// TIA Portal V20 export
// export: Created 2025-12-01T14:57:12.2354919Z, ExportSetting None, DisplayName Totally Integrated Automation Portal, DisplayVersion V20 Update 3, DisplayName TIA Portal Openness, DisplayVersion V20 Update 3, DisplayName TIA Portal Version Control Interface, DisplayVersion V20 Update 3, DisplayName STEP 7 Professional, DisplayVersion V20 Update 3, DisplayName STEP 7 Safety, DisplayVersion V20 Update 2, DisplayName WinCC Basic/Comfort/Advanced, DisplayVersion V20 Update 3, DisplayName WinCC Professional, DisplayVersion V20 Update 3, DisplayName WinCC Unified, DisplayVersion V20 Update 3
FUNCTION "FC993_CTRL_VAR_Lenze_i550_ASi" : Void   // FC993, LAD
{ S7_Optimized_Access := 'TRUE' }
// M.Familiar: Adaptado al nuevo base 14_02_2023.
// stored: AutoNumber false, SetENOAutomatically false
   VAR_INPUT
      DIR_INI_NODO : Int;   // Direccion inicial Gateway
      Num_Motor : Int;   // Numero de motor
      Avance : Bool;
      Retroceso : Bool;
      Rearme : Bool;   // Rearme variador
      Conexion_Estrella : Bool;
      Motor_2 : Bool;
      Sentido_Giro : Bool;   // Sentido giro
      "Activar Salida Digital DO1" : Bool;   // Activar Salida DO1
      Consigna_FR : Word;   // Consigna
   END_VAR
   VAR_TEMP
      ByteOffset : Int;
      Codigo_Area_Lectura : Byte;
      Codigo_Area_Escritura : Byte;
      Byte1_Status_Variador : Byte;
      Byte2_Status_Variador : Byte;
      Byte1PalabraControl : Byte;
      Byte2PalabraControl : Byte;
      Num_SETUP : Int;   // 1-triangulo Motor1/ 2-triangulo Motor 2 / 3-Estrella Motor1/4-Estrella Motor 2
   END_VAR
   VAR CONSTANT
      Area_SCR_DB : Byte := 16#84;
   END_VAR
BEGIN

REGION Network 1 (SCL): Simulador on?
   IF "Activar_Simulador" THEN
       #Codigo_Area_Lectura := 16#81;     // Area entradas %I
       #Codigo_Area_Escritura := 16#82;  // Area salidas %Q
   ELSE
       #Codigo_Area_Lectura := 16#1;     // Area entradas periferia 
       #Codigo_Area_Escritura := 16#2;  // Area salidas periferia 
   END_IF;
END_REGION

REGION Network 2 (SCL): Calcular Direccion inicial del nodo
   // M.FAMILIAR : Cambio calculo inicial de Byteoffset en base a direccion inicial de GATEWAY por directamnete direccion inicial del nodo del motor.
   REGION  //Definicion de direcciones a tratar//
       #ByteOffset := #DIR_INI_NODO;   

   END_REGION
END_REGION

REGION Network 3 (SCL): Lectura variador >>PLC
   REGION // lectura Status Variador    

       #Byte2_Status_Variador := PEEK_BYTE(area := #Codigo_Area_Lectura, dbNumber := 0, byteOffset := #ByteOffset);  //Leemos segundo Byte del status variador.
       POKE(area := #Area_SCR_DB,                                //Definimos tipo de area de memoria de escritura, en este caso un DB.
            dbNumber := 941,                                    //Ponemos 0 si es area de E/S si no ponemos numero de DB.
            byteOffset := (#Num_Motor * 18 - 17),                  // Definimos offset de Byte donde queremos escribir.
            value := #Byte2_Status_Variador,                 // valor que queremos escribir en destino.
            ENO => ENO);                                       // Consulta de ejecucion.
       #Byte1_Status_Variador := PEEK_BYTE(area := #Codigo_Area_Lectura, dbNumber := 0, byteOffset := #ByteOffset+1);  //Leemos primer Byte del status variador.
       POKE(area := #Area_SCR_DB,                                //Definimos tipo de area de memoria de escritura, en este caso un DB.
            dbNumber := 941,                                    //Ponemos 0 si es area de E/S si no ponemos numero de DB.
            byteOffset := (#Num_Motor* 18 - 18),                  // Definimos offset de Byte donde queremos escribir.
            value := #Byte1_Status_Variador,                 // valor que queremos escribir en destino.
            ENO => ENO);





    //lectura Words de codigo de error y corriente actual motor

       "DB941_Datos_VAR_Lenze_i550_ASi".Lenze_i550[#Num_Motor]."Código de error (Inputs)" := PEEK_WORD (area := #Codigo_Area_Lectura, dbNumber := 0, byteOffset := #ByteOffset + 2);
       "DB941_Datos_VAR_Lenze_i550_ASi".Lenze_i550[#Num_Motor]."Corriente actual (Inputs)" := PEEK_WORD (area := #Codigo_Area_Lectura, dbNumber := 0, byteOffset := #ByteOffset + 4);

    END_REGION
END_REGION

REGION Network 4 (SCL): Seleccion de SetUp Motor
   REGION Selección de juego de parámetros


       // SETUP 1__MOTOR 1 EN "TRIANGULO"
       IF (NOT #Conexion_Estrella AND NOT #Motor_2)
       THEN
           #Num_SETUP := 1;
       END_IF;


       // SETUP 2__MOTOR 2 EN "TRIANGULO"
       IF (NOT #Conexion_Estrella AND #Motor_2)
       THEN
           #Num_SETUP := 2;
       END_IF;


       // SETUP 3__MOTOR 1 EN "ESTRELLA"
       IF (#Conexion_Estrella AND NOT #Motor_2)
       THEN
           #Num_SETUP := 3;
       END_IF;


       // SETUP 4__MOTOR 2 EN "ESTRELLA"
       IF (#Conexion_Estrella AND #Motor_2)
       THEN
           #Num_SETUP := 4;
       END_IF;


   END_REGION




   REGION Ejecución de juego de parámetros

      CASE #Num_SETUP OF
           1:  // SETUP 1  triangulo motor 1 SETUP1
               "DB941_Datos_VAR_Lenze_i550_ASi".Lenze_i550[#Num_Motor]."Palabra de control (Outputs)"."Sel. paramset b0" := FALSE;
               "DB941_Datos_VAR_Lenze_i550_ASi".Lenze_i550[#Num_Motor]."Palabra de control (Outputs)"."Sel. paramset b1" := FALSE;
               ;
           2:  // SETUP 2  triangulo motor 2 SETUP2
               "DB941_Datos_VAR_Lenze_i550_ASi".Lenze_i550[#Num_Motor]."Palabra de control (Outputs)"."Sel. paramset b0" := TRUE;
               "DB941_Datos_VAR_Lenze_i550_ASi".Lenze_i550[#Num_Motor]."Palabra de control (Outputs)"."Sel. paramset b1" := FALSE;
               ;
           3:   // SETUP 3  estrella motor 1 SETUP3
               "DB941_Datos_VAR_Lenze_i550_ASi".Lenze_i550[#Num_Motor]."Palabra de control (Outputs)"."Sel. paramset b0" := FALSE;
               "DB941_Datos_VAR_Lenze_i550_ASi".Lenze_i550[#Num_Motor]."Palabra de control (Outputs)"."Sel. paramset b1" := TRUE;
               ;
          4:   // SETUP 4  estrella motor 2 SETUP4
               "DB941_Datos_VAR_Lenze_i550_ASi".Lenze_i550[#Num_Motor]."Palabra de control (Outputs)"."Sel. paramset b0" := TRUE;
               "DB941_Datos_VAR_Lenze_i550_ASi".Lenze_i550[#Num_Motor]."Palabra de control (Outputs)"."Sel. paramset b1" := TRUE;
               ;
          ELSE  // Si se mete un valor diferente se usa SETUP1
               "DB941_Datos_VAR_Lenze_i550_ASi".Lenze_i550[#Num_Motor]."Palabra de control (Outputs)"."Sel. paramset b0" := FALSE;
               "DB941_Datos_VAR_Lenze_i550_ASi".Lenze_i550[#Num_Motor]."Palabra de control (Outputs)"."Sel. paramset b1" := FALSE;
               ;
       END_CASE;
   END_REGION
END_REGION

REGION Network 5 (SCL): Ejecución de la función

   REGION //Region Control marcha/paro/direccion//
       //Region Control marcha/paro/direccion//

       IF ("DB941_Datos_VAR_Lenze_i550_ASi".Lenze_i550[#Num_Motor]."Estatus variador (Inputs)"."Ready for operation" AND  //Si ready for operation//
           "DB941_Datos_VAR_Lenze_i550_ASi".Lenze_i550[#Num_Motor]."Estatus variador (Inputs)"."Auto setp active" AND      //Si auto setpoint active//     
           NOT "DB941_Datos_VAR_Lenze_i550_ASi".Lenze_i550[#Num_Motor]."Estatus variador (Inputs)"."Fault active") THEN    // si no hay error activo//

           "DB941_Datos_VAR_Lenze_i550_ASi".Lenze_i550[#Num_Motor]."Error activo" := true;                // Activamos Condiciones OK//


           IF (#Avance AND NOT #Retroceso AND NOT #Sentido_Giro)OR ( #Sentido_Giro AND #Retroceso AND NOT #Avance) THEN
               "DB941_Datos_VAR_Lenze_i550_ASi".Lenze_i550[#Num_Motor]."Consigna de frecuencia (Outputs)" := #Consigna_FR;
               "DB941_Datos_VAR_Lenze_i550_ASi".Lenze_i550[#Num_Motor]."Palabra de control (Outputs)"."Run forward" := true;


           ELSE
               IF (NOT #Avance AND #Retroceso AND NOT #Sentido_Giro) OR (#Sentido_Giro AND NOT #Retroceso AND #Avance) THEN
                   "DB941_Datos_VAR_Lenze_i550_ASi".Lenze_i550[#Num_Motor]."Consigna de frecuencia (Outputs)" := #Consigna_FR;
                   "DB941_Datos_VAR_Lenze_i550_ASi".Lenze_i550[#Num_Motor]."Palabra de control (Outputs)"."Run forward" := true;
                   "DB941_Datos_VAR_Lenze_i550_ASi".Lenze_i550[#Num_Motor]."Palabra de control (Outputs)"."Reverse rotation dirtect." := true;


               ELSE
                   "DB941_Datos_VAR_Lenze_i550_ASi".Lenze_i550[#Num_Motor]."Consigna de frecuencia (Outputs)" := 0;
                   "DB941_Datos_VAR_Lenze_i550_ASi".Lenze_i550[#Num_Motor]."Palabra de control (Outputs)"."Run forward" := false;
                   "DB941_Datos_VAR_Lenze_i550_ASi".Lenze_i550[#Num_Motor]."Palabra de control (Outputs)"."Reverse rotation dirtect." := false;
               END_IF;

           END_IF;
       ELSE
           "DB941_Datos_VAR_Lenze_i550_ASi".Lenze_i550[#Num_Motor]."Error activo" := false;          //Si no se cumplen condiciones, descativamos condiciones OK//

       END_IF;
   END_REGION

   REGION  //Region Rearme//
       //Region Rearme//

       IF (#Rearme) THEN
           "DB941_Datos_VAR_Lenze_i550_ASi".Lenze_i550[#Num_Motor]."Palabra de control (Outputs)"."Reset error" := True;
       ELSE
           "DB941_Datos_VAR_Lenze_i550_ASi".Lenze_i550[#Num_Motor]."Palabra de control (Outputs)"."Reset error" := false;
       END_IF;
   END_REGION

   REGION // Activar salida DO1

       IF #"Activar Salida Digital DO1" THEN
           "DB941_Datos_VAR_Lenze_i550_ASi".Lenze_i550[#Num_Motor]."Palabra de control (Outputs)"."Activar salida DO1" := True;
       ELSE
           "DB941_Datos_VAR_Lenze_i550_ASi".Lenze_i550[#Num_Motor]."Palabra de control (Outputs)"."Activar salida DO1" := false;
       END_IF;
   END_REGION
END_REGION

REGION Network 6 (SCL): Escitura PLC>>Variador
   REGION
       REGION //Condiciones OK//

           IF  ("DB941_Datos_VAR_Lenze_i550_ASi".Lenze_i550[#Num_Motor]."Estatus variador (Inputs)"."Ready for operation" AND

               "DB941_Datos_VAR_Lenze_i550_ASi".Lenze_i550[#Num_Motor]."Estatus variador (Inputs)"."Auto setp active" AND

        NOT    "DB941_Datos_VAR_Lenze_i550_ASi".Lenze_i550[#Num_Motor]."Estatus variador (Inputs)"."Fault active") THEN

               "DB941_Datos_VAR_Lenze_i550_ASi".Lenze_i550[#Num_Motor]."Error activo" := FALSE;

           ELSE

               "DB941_Datos_VAR_Lenze_i550_ASi".Lenze_i550[#Num_Motor]."Error activo" := TRUE;
           END_IF;
       END_REGION

   END_REGION


   REGION //Escritura palabra de control//
       //Region escritura palabra de control//
       #Byte1PalabraControl := PEEK_BYTE(area := #Area_SCR_DB, dbNumber := 941, byteOffset := (#Num_Motor * 18 - 12));
       POKE(area := #Codigo_Area_Escritura,                                           //Definimos tipo de area de memoria de escritura, es salida o salida de periferia.
            dbNumber := 0,                                                           //Ponemos 0 si es area de E/S si no ponemos numero de DB.
            byteOffset := #ByteOffset +1,                                          // Definimos offset de Byte donde queremos escribir.
            value := #Byte1PalabraControl,                                         // valor que queremos escribir en destino.
            ENO => ENO);
       #Byte2PalabraControl := PEEK_BYTE(area := #Area_SCR_DB, dbNumber := 941, byteOffset := (#Num_Motor * 18 - 11));
       POKE(area := #Codigo_Area_Escritura,                                           //Definimos tipo de area de memoria de escritura, es salida o salida de periferia.
            dbNumber := 0,                                                           //Ponemos 0 si es area de E/S si no ponemos numero de DB.
            byteOffset := #ByteOffset ,                                          // Definimos offset de Byte donde queremos escribir.
            value := #Byte2PalabraControl,                                         // valor que queremos escribir en destino.
            ENO => ENO);

   END_REGION

   REGION
       // Escritura Words, Consigna y deceleracion// 
       POKE(area := #Codigo_Area_Escritura,                                           //Definimos tipo de area de memoria de escritura, es salida o salida de periferia.
            dbNumber := 0,                                                           //Ponemos 0 si es area de E/S si no ponemos numero de DB.
            byteOffset := #ByteOffset + 2,                                          // Definimos offset de Byte donde queremos escribir.
            value := "DB941_Datos_VAR_Lenze_i550_ASi".Lenze_i550[#Num_Motor]."Consigna de frecuencia (Outputs)");     // valor que queremos escribir en destino.

       POKE(area := #Codigo_Area_Escritura,                                       //Definimos tipo de area de memoria de escritura, es salida o salida de periferia.
            dbNumber := 0,                                                       //Ponemos 0 si es area de E/S si no ponemos numero de DB.
            byteOffset := #ByteOffset + 4,                                      // Definimos offset de Byte donde queremos escribir.
            value := "DB941_Datos_VAR_Lenze_i550_ASi".Lenze_i550[#Num_Motor]."DCC (Outputs)");                      // valor que queremos escribir en destino.
   END_REGION
END_REGION
END_FUNCTION
